FUNCTION_BLOCK E_SPLIT (* Split one event into two events *)
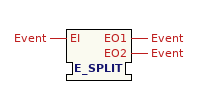
  EVENT_INPUT
    EI; (* Input event *)
  END_EVENT
  EVENT_OUTPUT
    EO1; (* First output event *)
    EO2; (* Second output event *)
  END_EVENT
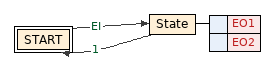
  EC_STATES
    START; (* Initial State *)
    State : -> EO1, -> EO2; (* Output events *)
  END_STATES
  EC_TRANSITIONS
    START TO State := EI;
    State TO START := 1;
  END_TRANSITIONS
END_FUNCTION_BLOCK
